// TIA Portal V16 export
// export: Created 2023-10-30T22:43:55.8067617Z, ExportSetting WithDefaults, DisplayName Totally Integrated Automation Portal, DisplayVersion V16, DisplayName TIA Portal Version Control Interface, DisplayVersion V16, DisplayName TIA Portal Openness, DisplayVersion V16, DisplayName SINAMICS Startdrive Advanced, DisplayVersion V16, DisplayName SINAMICS Startdrive G130, G150, S120, S150, SINAMICS MV, S210, DisplayVersion V16, DisplayName SINAMICS Startdrive G110M, G120, G120C, G120D, G120P, DisplayVersion V16, DisplayName STEP 7 Professional, DisplayVersion V16, DisplayName STEP 7 Safety, DisplayVersion V16, DisplayName WinCC Professional, DisplayVersion V16
DATA_BLOCK "Conversor_4-20_0-20_DB_1"   // DB22
VERSION : 0.1
// stored: AutoNumber true, DBAccessibleFromOPCUA true, InstanceOfName Conversor_4-20_0-20, InstanceOfType FB
"Conversor_4-20_0-20"
   // VAR_INPUT
   //    "IN_4-20" : Word;
   // END_VAR
   // VAR_OUTPUT
   //    "OUT_0-20" : Real;
   // END_VAR
BEGIN
END_DATA_BLOCK
